FUNCTION_BLOCK FB_CycleMan
VAR_INPUT
	xStart : BOOL;
	xStop : BOOL;
	
	
END_VAR
VAR_OUTPUT
	fbRtrigStart:R_trig;
	xBusy:BOOL;
	iEtape:INT;
END_VAR
VAR
	fbEtape:FB_Etape;
	inc: INT;
END_VAR

fbEtape.mActualisation(FALSE,FALSE);

fbRtrigStart(clk:=fbBtn.xStart);


CASE fbEtape.iNo OF
	0:	fbEtape.psMess:='Manual | Wait';
		IF xStart THEN
			fbEtape.piVal:=100;
		END_IF
	100:fbEtape.psMess:='Manual | Select what to do';
		//changer de mode
		IF  stParam.stStatus.eMMA<>Man THEN
			fbEtape.piSVal:=990;
		END_IF
		//Act1:
		IF (fbBtn.xManualAct1GoIn) THEN
			fbEtape.piVal:=201;
		END_IF
		IF (fbBtn.xManualAct1GoOut) THEN
			fbEtape.piVal:=202;
		END_IF
		IF fbBtn.xSetHomePos THEN
			fbEtape.piVal:=300;
		END_IF
		
		
		
		
	201: fbEtape.psMess:='Manual | Action : Act 1 Go in';
		IF (NOT fbBtn.xManualAct1GoIn) THEN
			fbEtape.piVal:=100;
		END_IF
	202: fbEtape.psMess:='Manual | Action : Act 1 Go out';
		IF (NOT fbBtn.xManualAct1GoOut) THEN
			fbEtape.piVal:=100;
		END_IF
	300: fbEtape.psMess:='Manual | Set Home Position';
		stParam.stMachine.stPosition0.Initialized:=TRUE;
		stParam.stMachine.stPosition0.PosX:=fbMotorX.fbAxisRef.NcToPlc.ActPos;
		stParam.stMachine.stPosition0.PosY:=fbMotorY.fbAxisRef.NcToPlc.ActPos;
		fbEtape.piVal:=100;
	
	990:fbEtape.psMess:='Manual | Finishing';
		//ici on fait des choses de fin (ex. eteindre un Motor qui tourne encore)
		IF (1) THEN
			fbEtape.piSVal:=999;
		END_IF	
	999:fbEtape.psMess:='Manual | Finished';
		IF (xStop) THEN
			fbEtape.piSVal:=0;
		END_IF
		
END_CASE

xBusy:=fbEtape.iNo<>0;
iEtape:=fbEtape.iNo;

END_FUNCTION_BLOCK

(* stored: Version 1.1.0.1, ProductVersion 3.1.4020.12
   POU FB_CycleMan: Id {0a4059b2-71e6-4341-9059-42714db8bec8}, SpecialFunc None *)
